// TIA Portal V17 export
// export: Created 2025-06-26T06:49:15.5430095Z, ExportSetting WithDefaults, DisplayName Totally Integrated Automation Portal, DisplayVersion V17 Update 8, DisplayName TIA Portal Openness, DisplayVersion V17 Update 8, DisplayName TIA Portal Version Control Interface, DisplayVersion V17, DisplayName STEP 7 Professional, DisplayVersion V17 Update 8, DisplayName STEP 7 Safety, DisplayVersion V17 Update 6, DisplayName WinCC Advanced, DisplayVersion V17 Update 8
FUNCTION_BLOCK "fbNullRegulator"   // FB59, FBD
TITLE = PI Regulator
{ S7_Optimized_Access := 'TRUE' }
VERSION : 0.1
// stored: AutoNumber true, IsIECCheckEnabled false, IsRetainMemResEnabled false, MemoryReserve 0, SetENOAutomatically false, UDAEnableTagReadback false
   VAR_INPUT
      bEnable : Bool;
      bReset : Bool;
   END_VAR
   VAR_OUTPUT
      fOut : Real;
      bAtMin : Bool;
      bAtMax : Bool;
   END_VAR
   VAR_IN_OUT
      sTag : "stNullRegulator";
   END_VAR
   VAR
      Dummy : Real;
   END_VAR
   VAR_TEMP
      Enabled : Bool;
      fSelectedSetpoint : Real;
   END_VAR
BEGIN

REGION Network 1: Reset manual mode
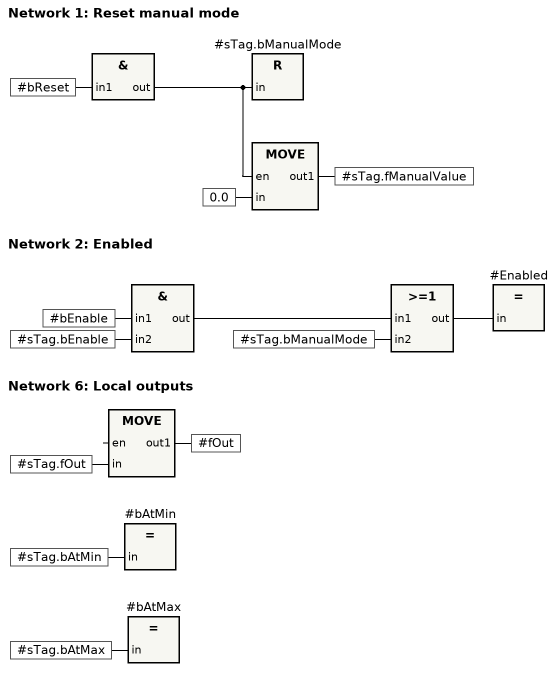
   IF #bReset THEN
       #sTag.bManualMode := FALSE;
       #sTag.fManualValue := 0.0;
   END_IF;
END_REGION

REGION Network 2: Enabled
   // Local input is from process control logic: when to run the regulator
   // Tag input is from HMI: do we want to run this regulator at all
   #Enabled := (#bEnable AND #sTag.bEnable) OR #sTag.bManualMode;
END_REGION

REGION Network 3 (SCL): Output selection
   IF #sTag.bManualMode = TRUE THEN
       #fSelectedSetpoint := #sTag.fManualValue;
   ELSE
       #fSelectedSetpoint := #sTag.fSetpoint;
   END_IF;

   #sTag.fOut := LIMIT(MN := #sTag.fOutMin, IN := #fSelectedSetpoint, MX := #sTag.fOutMax);
   #sTag.bAtMin := #sTag.fOut = #sTag.fOutMin;
   #sTag.bAtMax := #sTag.fOut = #sTag.fOutMax;
END_REGION

REGION Network 4 (SCL): Disable
   // This could be combined with logic above, and one day it might be!
   IF #Enabled = FALSE OR #sTag.bFault = TRUE THEN
       #sTag.fOut := 0.0;
       #sTag.bAtMin := FALSE;
       #sTag.bAtMax := FALSE;
   END_IF;
END_REGION

REGION Network 5 (SCL): Mode
   // Mode
   IF #sTag.bManualMode = TRUE THEN
       #sTag.nMode := 2;
   ELSIF #sTag.bEnable = TRUE THEN
       #sTag.nMode := 1;
   ELSE
       #sTag.nMode := 0;
   END_IF;
END_REGION

REGION Network 6: Local outputs
   #fOut := #sTag.fOut;
   #bAtMin := #sTag.bAtMin;
   #bAtMax := #sTag.bAtMax;
END_REGION
END_FUNCTION_BLOCK
